PROGRAM prgCS
VAR
	fbRTUMaster					: FB_KL6xxx_ModbusRTU_22B_Master;
	byErrorwarningRTU			: BYTE;									//{#lynus.ag#()}
	fbCS1						: FB_ECS_Schrack_EM_CionHome;			//{#lynus.ag#()}
	fbCS2						: FB_ECS_Schrack_EM_CionHome;			//{#lynus.ag#()}
	fbCS3						: FB_ECS_Schrack_EM_CionHome;			//{#lynus.ag#()}
	bCarConnCS1					: BOOL;									//{#lynus.ag#()}
	bCarConnCS2					: BOOL;									//{#lynus.ag#()}
	bCarConnCS3					: BOOL;									//{#lynus.ag#()}
	bOnEmergPowerOffCS1			: BOOL;									//{#lynus.ag#()}
	bOnEmergPowerOffCS2			: BOOL;									//{#lynus.ag#()}
	bOnEmergPowerOffCS3			: BOOL;									//{#lynus.ag#()}
	bSOnEmergPowerOffCS1		: BOOL;									//{#lynus.ag#()}
	bSOnEmergPowerOffCS2		: BOOL;									//{#lynus.ag#()}
	bSOnEmergPowerOffCS3		: BOOL;									//{#lynus.ag#()}
	byErrorWarningCS1			: BYTE;									//{#lynus.ag#()}
	byErrorWarningCS2			: BYTE;									//{#lynus.ag#()}
	byErrorWarningCS3			: BYTE;									//{#lynus.ag#()}
	wCPStateCS1					: WORD;									//{#lynus.ag#()}
	bChargingReleaseInavlidCS1	: BOOL;									//{#lynus.ag#()}
	rChargingTimeInMinCS1		: REAL;									//{#lynus.ag#()}
	wCPStateCS2					: WORD;									//{#lynus.ag#()}
	bChargingReleaseInavlidCS2	: BOOL;									//{#lynus.ag#()}
	rChargingTimeInMinCS2		: REAL;									//{#lynus.ag#()}
	wCPStateCS3					: WORD;									//{#lynus.ag#()}
	bChargingReleaseInavlidCS3	: BOOL;									//{#lynus.ag#()}
	rChargingTimeInMinCS3		: REAL;									//{#lynus.ag#()}
	byErrorCounter				: BYTE;									//{#lynus.ag#()}
	FpErrror					: R_TRIG;
END_VAR

//Power Data
//Each CS has 14kW

fbRTUMaster(
	bConfigTerminal:= , 
	uiKBusState_IN:= prgKNX.fbKBusState.uiKBusState_OUT, 
	bBusy=> , 
	byErrorWarning=> , 
	byActualAdressInUse=> , 
	diNrOfMBRTUMasterLine_OUT=> , 
	eMessageMBRTUMaster=> , 
	bTerminalIsConfigured=> );

fbRTUMaster(
	bConfigTerminal:= , 
	bBusy=> , 
	byErrorWarning=> , 
	diNrOfMBRTUMasterLine_OUT=> , 
	eMessageMBRTUMaster=> , 
	bTerminalIsConfigured=> );

byErrorwarningRTU := fbRTUMaster.byErrorWarning;

FpErrror(CLK:= byErrorwarningRTU = 2, Q=> );
	IF FpErrror.Q THEN byErrorCounter := byErrorCounter + 1; END_IF
	
//Garage 1 near Door	
fbCS1.stSetupECS.bOnEmergPowerOff := bOnEmergPowerOffCS1;

fbCS1(
	bEnable:= , 
	bPowerDataInvers:= , 
	byMBAdress:= 1, 
	diNrOfMBRTUMasterLine_IN:= fbRTUMaster.diNrOfMBRTUMasterLine_OUT, 
	diNrOfEMS_IN:= prgEMS.EMS.diNrOfEMS_OUT, 
	diNrOfEM_IN_CS:= , 
	stSetupECS:= , 
	stDataECS=> , 
	eSchrackErrors=> , 
	diNrOfECS_OUT=> );

wCPStateCS1:= fbCS1.wCPStateECS;
	bChargingReleaseInavlidCS1 := fbCS1.bChargingReleaseInavlid;
		rChargingTimeInMinCS1 := fbCS1.stDataECS.arrChargingTimeInMin[1];
			byErrorWarningCS1 := fbCS1.stDataECS.byErrorWarning;
				bCarConnCS1 := fbCS1.stDataECS.bCarConnected;
					bSOnEmergPowerOffCS1 := fbCS1.stDataECS.bSOnEmergPowerOff;
	
//Between CS1	
fbCS2.stSetupECS.bOnEmergPowerOff := bOnEmergPowerOffCS2;

fbCS2(
	bEnable:= , 
	bPowerDataInvers:= , 
	byMBAdress:= 2, 
	diNrOfMBRTUMasterLine_IN:= fbRTUMaster.diNrOfMBRTUMasterLine_OUT, 
	diNrOfEMS_IN:= prgEMS.EMS.diNrOfEMS_OUT, 
	diNrOfEM_IN_CS:= , 
	stSetupECS:= , 
	stDataECS=> , 
	eSchrackErrors=> , 
	diNrOfECS_OUT=> );

wCPStateCS2:= fbCS2.wCPStateECS;
	bChargingReleaseInavlidCS2 := fbCS2.bChargingReleaseInavlid;
		rChargingTimeInMinCS2 := fbCS2.stDataECS.arrChargingTimeInMin[1];
			byErrorWarningCS2 := fbCS2.stDataECS.byErrorWarning;
				bCarConnCS2 := fbCS2.stDataECS.bCarConnected;
					bSOnEmergPowerOffCS2 := fbCS2.stDataECS.bSOnEmergPowerOff;	
	
//Outdoor CS
fbCS3.stSetupECS.bOnEmergPowerOff := bOnEmergPowerOffCS3;

fbCS3(
	bEnable:= , 
	bPowerDataInvers:= , 
	byMBAdress:= 3, 
	diNrOfMBRTUMasterLine_IN:= fbRTUMaster.diNrOfMBRTUMasterLine_OUT, 
	diNrOfEMS_IN:= prgEMS.EMS.diNrOfEMS_OUT, 
	diNrOfEM_IN_CS:= , 
	stSetupECS:= , 
	stDataECS=> , 
	eSchrackErrors=> , 
	diNrOfECS_OUT=> );
	
wCPStateCS3:= fbCS3.wCPStateECS;
	bChargingReleaseInavlidCS3 := fbCS3.bChargingReleaseInavlid;
		rChargingTimeInMinCS3 := fbCS3.stDataECS.arrChargingTimeInMin[1];
			byErrorWarningCS3 := fbCS3.stDataECS.byErrorWarning;
				bCarConnCS3 := fbCS3.stDataECS.bCarConnected;
					bSOnEmergPowerOffCS3 := fbCS3.stDataECS.bSOnEmergPowerOff;

END_PROGRAM

(* stored: Version 1.1.0.1, ProductVersion 3.1.4024.9
   POU prgCS: Id {59551682-60c0-4b8c-b147-ae376642129b}, SpecialFunc None *)
